(* PLC project  *)

CONFIGURATION Robot_A
END_CONFIGURATION
